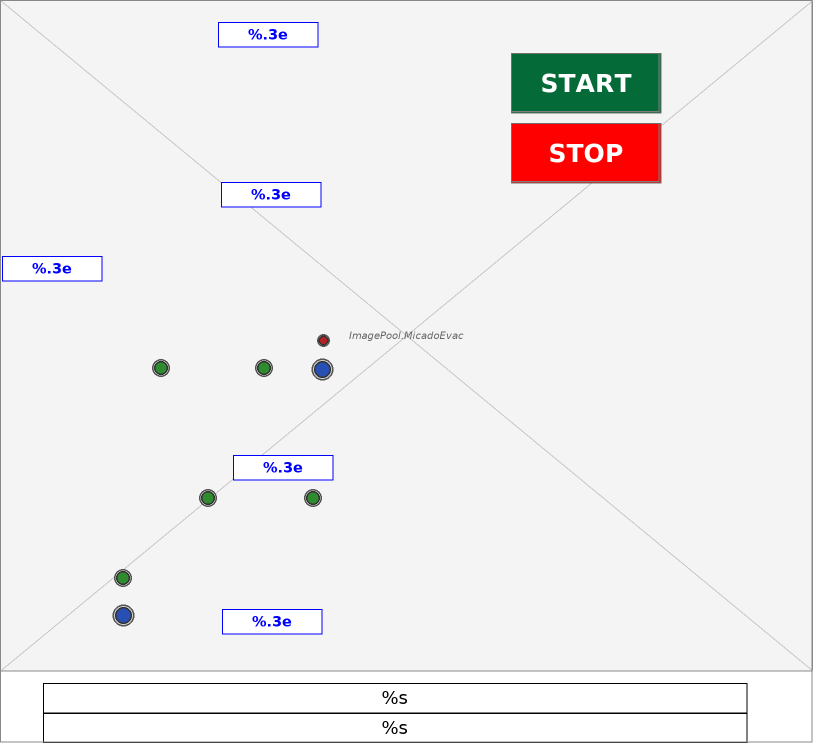
VISUALIZATION GUI_EVAC_MICADO  // 813x743
    Image (0,0 813x671), image: ImagePool.MicadoEvac
    Rectangle (222,609 100x25), "%.3e", text variable: MAIN.evac_micado.VAG1.stat.lrPressure
    Rectangle (233,455 100x25), "%.3e", text variable: MAIN.evac_micado.VAG2.stat.lrPressure
    Rectangle (2,256 100x25), "%.3e", text variable: MAIN.evac_micado.VAG3.stat.lrPressure
    Rectangle (218,22 100x25), "%.3e", text variable: MAIN.evac_micado.VAGF.stat.lrPressure
    Rectangle (221,182 100x25), "%.3e", text variable: MAIN.evac_micado.VAGG.stat.lrPressure
    Lamp1 (111,603 25x25), variable: MAIN.evac_micado.rp.stat.bReady, style: Lamp-Lamp1-Blue
    Lamp1 (310,357 25x25), tooltip "If ON, TMP pump is at its nominal speed, i.e. Ready.", variable: MAIN.evac_micado.tp.stat.bReady, style: Lamp-Lamp1-Blue
    Lamp1 (198,488 20x20), variable: MAIN.evac_micado.PVV1.stat.bActON, style: Lamp-Lamp1-Green
    Lamp1 (303,488 20x20), variable: MAIN.evac_micado.PVV2.stat.bActON, style: Lamp-Lamp1-Green
    Lamp1 (151,358 20x20), variable: MAIN.evac_micado.PVV3.stat.bActON, style: Lamp-Lamp1-Green
    Lamp1 (254,358 20x20), variable: MAIN.evac_micado.PVV4.stat.bActON, style: Lamp-Lamp1-Green
    Lamp1 (113,568 20x20), variable: MAIN.evac_micado.GBV.stat.bActON, style: Lamp-Lamp1-Green
    Rectangle (43,683 704x30), "%s", text variable: MAIN.evac_micado.stat.sErrorText
    Rectangle (43,713 704x30), "%s", text variable: MAIN.evac_micado.stat.sStatus
    Button (511,53 150x60), "START"
        OnMouseClick: execute { MAIN.bEnable_evac_mic := TRUE; }
    Button (511,123 150x60), "STOP"
        OnMouseClick: execute { MAIN.bEnable_evac_mic := FALSE; }
    Lamp1 (316,333 15x15), tooltip "If ON, TMP pump is still spinning.", variable: MAIN.evac_micado.tp.stat.bSpeed100, style: Lamp-Lamp1-Red
END_VISUALIZATION

(* stored: Version 1.1.0.1, ProductVersion 3.1.4024.9
   Visu GUI_EVAC_MICADO: Id {b2a05de4-3454-4682-9605-1f5c20d3d681} *)
